{attribute 'OPC.UA.DA.StructuredType' := '1'}
FUNCTION_BLOCK FB_BaseMachine_1
VAR

	{attribute 'OPC.UA.DA' := '0'} 
	bBusy: BOOL := FALSE;
	{attribute 'OPC.UA.DA' := '1'} 
	bError: BOOL := FALSE;
	{attribute 'OPC.UA.DA' := '1'} 
	bEnable: BOOL := FALSE;
	{attribute 'OPC.UA.DA' := '1'} 
	eState: E_MachineState := E_MachineState.IDLE;
	{attribute 'OPC.UA.DA' := '1'} 
	{attribute 'OPC.UA.DA.StructuredType' := '1'}
	fbSequenceManager: FB_SequenceManager_1;
	{attribute 'OPC.UA.DA' := '0'} 
	aAllComponents: ARRAY[1..50] OF POINTER TO FB_BaseDevice;
	
	{attribute 'OPC.UA.DA' := '1'} 
	aErrors: ARRAY[1..20] OF ST_Alarm;	// raiseEvent() method updates Error1 / aErrors[1] only at the moment, must implement a ring buffer with error active checking for full functionality

	
END_VAR 

VAR_INPUT
	{attribute 'OPC.UA.DA' := '1'} 
	sID: STRING;  
	{attribute 'OPC.UA.DA' := '1'} 
	sDescr: STRING;
	{attribute 'OPC.UA.DA' := '1'} 
	nQtyComponents: INT;
END_VAR

METHOD devices_disable_All : BOOL
VAR
	iterator: INT;
	
END_VAR
FOR iterator:=1 TO nQtyComponents BY 1 DO
	aAllComponents[iterator]^.disable();
END_FOR
END_METHOD

METHOD devices_disable_CurrSeq : BOOL
VAR
	iterator: INT;
	Steps : ARRAY[1..20] OF ST_SequenceStep;
END_VAR
FOR iterator:=1 TO fbSequenceManager.getCurrentSeq_FB()^.stepsTotal() BY 1 DO
	
	Steps := fbSequenceManager.getCurrentSeq_FB()^.steps();
	Steps[iterator].Device^.disable();
	
END_FOR
END_METHOD

METHOD devices_enable_All : BOOL
VAR
	iterator: INT;
END_VAR
FOR iterator:=1 TO nQtyComponents BY 1 DO
	aAllComponents[iterator]^.enable();
END_FOR
END_METHOD

METHOD devices_enable_CurrSeq : BOOL
VAR
	iterator: INT;
	Steps : ARRAY[1..20] OF ST_SequenceStep;
END_VAR
FOR iterator:=1 TO fbSequenceManager.getCurrentSeq_FB()^.stepsTotal() BY 1 DO
	Steps := fbSequenceManager.getCurrentSeq_FB()^.steps();
	Steps[iterator].Device^.enable();
END_FOR
END_METHOD

METHOD devices_setAuto_All : BOOL
VAR
	iterator: INT;
END_VAR
FOR iterator:=1 TO nQtyComponents BY 1 DO
	aAllComponents[iterator]^.setMode(Mode := E_DeviceMode.AUTO);
END_FOR
END_METHOD

METHOD devices_setAuto_CurrSeq : BOOL
VAR
	iterator: INT;
	Steps : ARRAY[1..20] OF ST_SequenceStep;
END_VAR
FOR iterator:=1 TO fbSequenceManager.getCurrentSeq_FB()^.stepsTotal() BY 1 DO
	
	Steps := fbSequenceManager.getCurrentSeq_FB()^.steps();
	Steps[iterator].Device^.setMode(Mode := E_DeviceMode.AUTO);
END_FOR
END_METHOD

METHOD devices_setManual_All : BOOL
VAR
	iterator: INT;
END_VAR
FOR iterator:=1 TO nQtyComponents BY 1 DO
	aAllComponents[iterator]^.setMode(Mode := E_DeviceMode.AUTO);
END_FOR
END_METHOD

METHOD devices_setManual_CurrSeq : BOOL
VAR
	iterator: INT;
	Steps : ARRAY[1..20] OF ST_SequenceStep;
END_VAR
FOR iterator:=1 TO fbSequenceManager.getCurrentSeq_FB()^.stepsTotal() BY 1 DO
	
	Steps := fbSequenceManager.getCurrentSeq_FB()^.steps();
	Steps[iterator].Device^.setMode(Mode := E_DeviceMode.MANUAL);
END_FOR
END_METHOD

METHOD seq_Pause : BOOL
VAR_INPUT
END_VAR
fbSequenceManager.pauseSequence();
END_METHOD

METHOD seq_Start : BOOL
VAR_INPUT
	SeqNum: UINT;
END_VAR
devices_disable_All();
fbSequenceManager.selectSequence(Sequence := 1);
devices_enable_CurrSeq();
fbSequenceManager.startSequence();
END_METHOD

METHOD seq_Stop : BOOL
VAR_INPUT
END_VAR
fbSequenceManager.stopSequence();
END_METHOD

END_FUNCTION_BLOCK

(* stored: Version 1.1.0.1, ProductVersion 3.1.4024.12
   POU FB_BaseMachine_1: Id {766a1d5a-77a4-42cb-9177-328046e9239a}, SpecialFunc None
   Method devices_disable_All: Id {23ddba9c-2992-470e-b20c-44df538fee1c}
   Method devices_disable_CurrSeq: Id {29da31d3-af10-4789-8902-00ef4038d748}
   Method devices_enable_All: Id {0838d4b0-fcb7-4cc9-844f-5213fad6845f}
   Method devices_enable_CurrSeq: Id {f05f6ed0-04bb-48f1-b8f1-83ebff03a6c8}
   Method devices_setAuto_All: Id {9e58380e-52f3-44c8-8f79-44f9e54b30ad}
   Method devices_setAuto_CurrSeq: Id {1eeb9fbf-5ca1-47dc-b2f7-7955ec2aef1b}
   Method devices_setManual_All: Id {791e8910-fbaf-4d87-b22f-ea88260b350d}
   Method devices_setManual_CurrSeq: Id {92db99d4-1d9f-4cc3-a9de-9884be5edc71}
   Method seq_Pause: Id {ec55b341-c13a-4a27-a9cd-881f229b0637}
   Method seq_Start: Id {fa42d325-30f5-4183-9428-8797d9f24688}
   Method seq_Stop: Id {4d5573eb-97a3-4b14-b23e-fc28b4b79496} *)
